FUNCTION_BLOCK SST_ControlOfOutputs
VAR_INPUT
END_VAR
VAR_OUTPUT
END_VAR
VAR
END_VAR

// NETWORK 1

END_FUNCTION_BLOCK

(* stored: Version 1.1.0.1, ProductVersion 3.1.4024.15
   POU SST_ControlOfOutputs: Id {d396a545-25be-4941-a2a8-8c39fe60fb6e}, SpecialFunc None *)
